(* CODESYS project test1.project

Project tree, tasks and I/O mapping:
  Device : CODESYS Control Win V3, 3S - Smart Software Solutions GmbH, order no. 305021, version 3.5.8.10
    application Application
      libraries: Standard, * (System)
      task MainTask (cyclic, interval t#20ms, priority 1) calls PLC_PRG
      task VISU_TASK (cyclic, interval 100 ms, priority 31) calls VisuElems.Visu_Prg
      program PLC_PRG [FBD]
      visualisation Visualization
  text list GlobalTextList
*)

// Device/Application/PLC_PRG
PROGRAM PLC_PRG
VAR
	t1: TON;
	zegar: BOOL;
	zmienna: TIME;
	
	przycisk1: BOOL;
	przycisk2: BOOL;
	przycisk3: BOOL;
	przycisk4: BOOL;
	przycisk5: BOOL;
	
	winda_na_1: BOOL;
	winda_na_5: BOOL;
	
	winda_1: BOOL;
	winda_5: BOOL;
	
	licznik: WORD;

	ctud1: CTUD;
	
	moveY: INT;
	
	nieaktywne: BOOL;

END_VAR

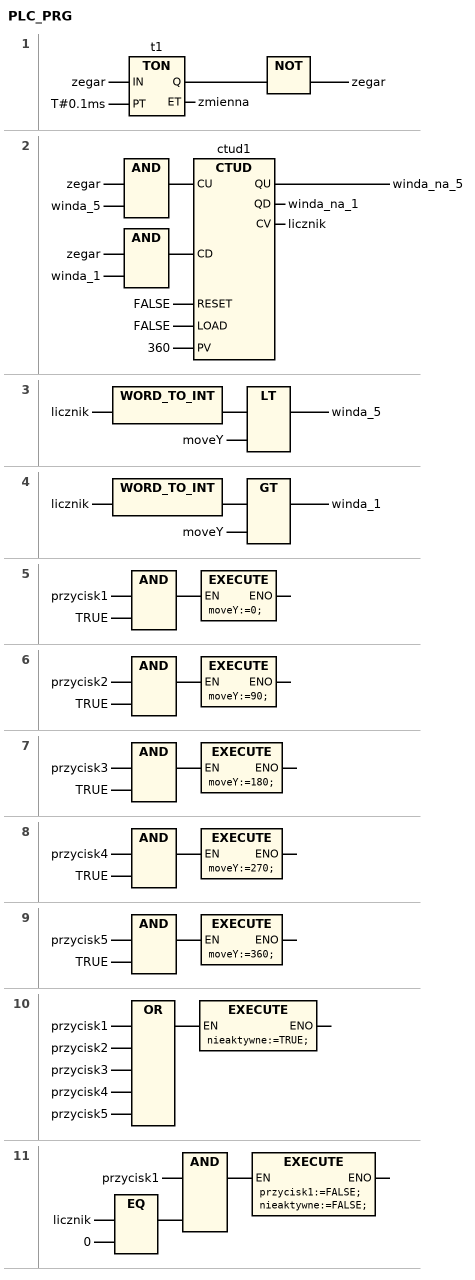
// NETWORK 1
t1(IN := zegar, PT := T#0.1ms, ET => zmienna); // TON
zegar := NOT t1.Q;

// NETWORK 2
ctud1(
    CU := zegar AND winda_5,
    CD := zegar AND winda_1,
    RESET := FALSE,
    LOAD := FALSE,
    PV := 360,
    QD => winda_na_1,
    CV => licznik); // CTUD
winda_na_5 := ctud1.QU;

// NETWORK 3
winda_5 := WORD_TO_INT(licznik) < moveY;

// NETWORK 4
winda_1 := WORD_TO_INT(licznik) > moveY;

// NETWORK 5
IF przycisk1 AND TRUE THEN moveY:=0; END_IF

// NETWORK 6
IF przycisk2 AND TRUE THEN moveY:=90; END_IF

// NETWORK 7
IF przycisk3 AND TRUE THEN moveY:=180; END_IF

// NETWORK 8
IF przycisk4 AND TRUE THEN moveY:=270; END_IF

// NETWORK 9
IF przycisk5 AND TRUE THEN moveY:=360; END_IF

// NETWORK 10
IF przycisk1 OR przycisk2 OR przycisk3 OR przycisk4 OR przycisk5 THEN nieaktywne:=TRUE; END_IF

// NETWORK 11
IF przycisk1 AND licznik = 0 THEN
    przycisk1:=FALSE;
    nieaktywne:=FALSE;
END_IF

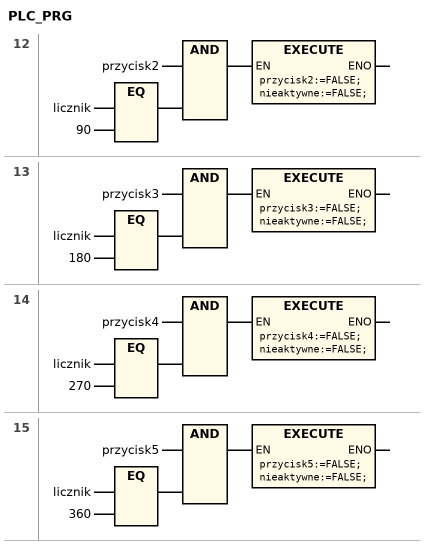
// NETWORK 12
IF przycisk2 AND licznik = 90 THEN
    przycisk2:=FALSE;
    nieaktywne:=FALSE;
END_IF

// NETWORK 13
IF przycisk3 AND licznik = 180 THEN
    przycisk3:=FALSE;
    nieaktywne:=FALSE;
END_IF

// NETWORK 14
IF przycisk4 AND licznik = 270 THEN
    przycisk4:=FALSE;
    nieaktywne:=FALSE;
END_IF

// NETWORK 15
IF przycisk5 AND licznik = 360 THEN
    przycisk5:=FALSE;
    nieaktywne:=FALSE;
END_IF

END_PROGRAM

// Device/Application/Visualization
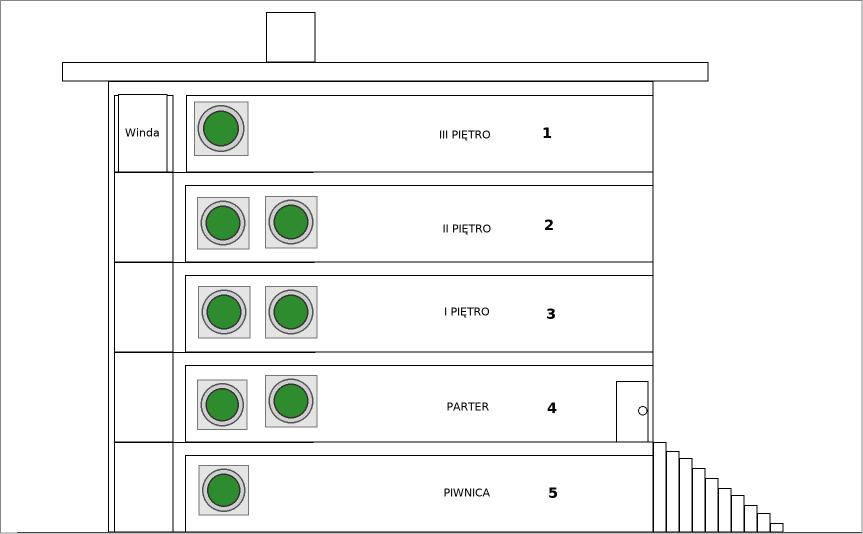
VISUALIZATION Visualization  // 863x534
    Rectangle (108,81 545x451)
    Rectangle (185,455 468x77)
    Rectangle (114,95 59x77)
    Rectangle (114,172 59x90)
    Rectangle (114,262 59x90)
    Rectangle (114,352 59x90)
    Rectangle (114,442 59x90)
    Rectangle (118,94 49x78), "Winda"
        p2738717112: PLC_PRG.licznik
    Rectangle (185,365 468x77)
    Rectangle (185,275 468x77)
    Rectangle (185,185 468x77)
    Rectangle (186,95 467x77)
    Rectangle (62,62 646x19)
    Rectangle (266,12 49x50)
    Line (662,532) (861,532)
    Rectangle (616,381 32x61)
    Rectangle (653,442 13x90)
    Rectangle (666,451 13x81)
    Rectangle (679,458 13x74)
    Rectangle (692,468 13x64)
    Rectangle (705,478 13x54)
    Rectangle (718,488 13x44)
    Rectangle (731,495 13x37)
    Rectangle (744,505 13x27)
    Rectangle (757,513 13x19)
    Rectangle (770,523 13x9)
    Line (17,532) (216,532)
    Line (114,442) (313,442)
    Line (116,352) (315,352)
    Line (115,262) (314,262)
    Line (114,172) (313,172)
    Ellipse (638,406 9x9)
    Label (392,478 150x30), "PIWNICA"
    Label (393,392 150x30), "PARTER"
    Label (392,297 150x30), "I PIĘTRO"
    Label (392,214 150x30), "II PIĘTRO"
    Label (390,120 150x30), "III PIĘTRO"
    PushSwitch (194,101 54x55), variable: PLC_PRG.przycisk1, input disabled if: PLC_PRG.nieaktywne, behaviour: TOGGLE, style: Switch-PushSwitch-Green
    PushSwitch (197,378 50x53), variable: PLC_PRG.przycisk4, input disabled if: PLC_PRG.nieaktywne, behaviour: TOGGLE, style: Switch-PushSwitch-Green
    PushSwitch (197,286 54x52), variable: PLC_PRG.przycisk3, input disabled if: PLC_PRG.nieaktywne, behaviour: TOGGLE, style: Switch-PushSwitch-Green
    PushSwitch (197,197 52x52), variable: PLC_PRG.przycisk2, input disabled if: PLC_PRG.nieaktywne, behaviour: TOGGLE, style: Switch-PushSwitch-Green
    PushSwitch (197,465 53x50), variable: PLC_PRG.przycisk5, input disabled if: PLC_PRG.nieaktywne, behaviour: TOGGLE, style: Switch-PushSwitch-Green
    PushSwitch (265,196 52x52), behaviour: TOGGLE, style: Switch-PushSwitch-Green
    PushSwitch (265,286 52x52), behaviour: TOGGLE, style: Switch-PushSwitch-Green
    PushSwitch (265,375 52x52), behaviour: TOGGLE, style: Switch-PushSwitch-Green
    Label (478,478 150x30), "5"
    Label (477,393 150x30), "4"
    Label (476,299 150x30), "3"
    Label (474,210 150x30), "2"
    Label (472,118 150x30), "1"
END_VISUALIZATION
